TYPE ST_Settings :
	STRUCT
		// Tenzo
		fTenzoCons   : LREAL := 0.01;
		fTenzoOffset : LREAL := 0.0; 
	
		// Force control
		fKp : LREAL := 10;
		fKi : LREAL := 0.1;
		fIntegralLimit  : LREAL := 10;
		fForceTolerance : LREAL := 0.1;
		fMaxVelocity    : LREAL := 100;
	
		// Motion safety
		fMaxForce    : LREAL := 10;
		fMaxPosition : LREAL := 0.1;
	END_STRUCT
END_TYPE

(* stored: Version 1.1.0.1, ProductVersion 3.1.4024.15
   DUT ST_settings: Id {4c7494d5-7e0d-4afe-afc6-07f6109539eb} *)
